PROGRAM MAIN
VAR
END_VAR

END_PROGRAM

(* stored: Version 1.1.0.1
   POU MAIN: Id {a1b4d7a7-30f6-4eca-9d8a-8886ed2e64bb} *)
